Yaskawa INFORM job: R1_W27-A3(90,0)OK-KM.JBI

/JOB
//NAME R1_W27-A3(90,0)OK-KM
///FOLDERNAME KRIS-SCIANA
//POS
///NPOS 39,39,0,3,0,0
///TOOL 0
///POSTYPE PULSE
///PULSE
C00000=28952,8585,-18317,-13996,70208,35679
C00001=71005,-6773,-21567,22823,106593,44775
C00002=117043,42996,63636,80074,76806,36548
C00003=119925,40522,60971,80546,74909,36908
C00004=120979,40510,60955,80742,74190,36976
C00005=121620,40526,60973,80863,73749,37016
C00006=120979,40510,60955,80742,74190,36976
C00007=120972,47430,68505,81028,73985,36463
C00008=120975,44790,65593,80913,74065,36669
C00009=119925,40522,60971,80546,74909,36908
C00010=117043,28525,29392,77595,79872,42812
C00011=119217,29213,30072,77642,78317,42963
C00012=118591,29142,41659,90629,77759,36862
C00013=119665,29075,41592,90781,76989,36871
C00014=118591,29142,41659,90629,77759,36862
C00015=119139,32499,45041,90778,77358,36699
C00016=118591,29142,41659,90629,77759,36862
C00017=117792,30891,31745,84274,86418,41418
C00018=115072,-13134,-7135,52375,63390,45207
C00019=116472,-2069,1649,51986,62773,45649
C00020=119056,6654,11865,54723,60280,45496
C00021=120221,1002,3727,51035,60853,46679
C00022=118976,344,2628,51184,61768,46509
C00023=114063,10407,25128,70575,62115,41682
C00024=112190,-3493,21544,75414,62330,39001
C00025=112095,-4963,21051,75629,62268,38767
C00026=109884,-10292,2975,62963,64916,42297
C00027=110682,-7799,62,53762,64868,43520
C00028=112905,-37925,-18654,59494,39923,-31745
C00029=119033,-32806,-15367,56336,36549,-29573
C00030=103409,10299,29788,79828,70646,-39016
C00031=118213,-31916,-14769,56613,37088,-29774
C00032=119040,-32554,-15197,56304,36559,-29555
C00033=101836,30280,52112,81952,79109,-40621
C00034=100971,47035,98169,91258,69327,-49643
C00035=93737,11259,49117,86061,72646,-45987
C00036=78961,-66055,-35758,60750,43436,-32907
C00037=20797,37541,-3335,35327,72696,-61186
C00038=29399,116943,32129,-7323,87105,-68619
BC00000=188265,1301853,894037
BC00001=296251,1242662,815779
BC00002=395849,1188070,743600
BC00003=395849,1188070,743600
BC00004=395849,1188070,743600
BC00005=395849,1188070,743600
BC00006=395849,1188070,743600
BC00007=395849,1188070,743600
BC00008=395849,1188070,743600
BC00009=395849,1188070,743600
BC00010=395849,1188070,743600
BC00011=395849,1188070,727654
BC00012=394310,1188070,721275
BC00013=394310,1188070,721275
BC00014=394310,1188070,721275
BC00015=394310,1188070,721275
BC00016=394310,1188070,721275
BC00017=395849,1177175,737022
BC00018=360898,1188070,902203
BC00019=357567,1188070,879539
BC00020=356337,1188069,883137
BC00021=356235,1188070,870473
BC00022=356235,1188070,870473
BC00023=356285,1188070,883286
BC00024=356285,1188070,883285
BC00025=356285,1188070,883285
BC00026=356318,1188070,883506
BC00027=360948,1188070,915014
BC00028=346658,1188070,806607
BC00029=342406,1188070,804445
BC00030=341079,1188070,803770
BC00031=340706,1188070,803580
BC00032=340706,1188070,803580
BC00033=340706,1188070,653450
BC00034=340706,1188070,803580
BC00035=341062,1188070,799461
BC00036=346492,1188070,736766
BC00037=227280,1187761,922106
BC00038=106915,1318361,1048473
///POSTYPE BASE
///RECTAN
///RCONF 0,0,0,0,0,0,0,0,0,0,0,0,0,0,0,0,0,0,0,0,0,0,0,0
P00006=0.222,-3.123,-1.508,0.0000,0.0000,0.0000
P00025=-2.003,0.006,0.728,0.0000,0.0000,0.0000
P00026=0.562,-0.002,-0.337,0.0000,0.0000,0.0000
//INST
///DATE 2024/07/29 20:46
///ATTR SC,RW
///GROUP1 RB1,BS1
NOP
SFTOF
MOVJ C00000 BC00000 VJ=100.00
MOVJ C00001 BC00001 VJ=100.00
MOVL C00002 BC00002 V=1000.0
MOVL C00003 BC00003 V=250.0
MOVL C00004 BC00004 V=100.0
REFP 3 C00005 BC00005
CALL JOB:SEARCH-R1
SET P026 P006
SFTON P026
MOVL C00006 BC00006 V=60.0
REFP 3 C00007 BC00007
CALL JOB:SEARCH-R1
SET P026 P006
SFTON P026
MOVL C00008 BC00008 V=60.0
MOVL C00009 BC00009 V=166.7
SFTOF
MOVL C00010 BC00010 V=1000.0
MOVL C00011 BC00011 V=250.0
MOVL C00012 BC00012 V=100.0
REFP 3 C00013 BC00013
CALL JOB:SEARCH-R1
SET P025 P006
SFTON P025
MOVL C00014 BC00014 V=100.0
REFP 3 C00015 BC00015
CALL JOB:SEARCH-R1
SET P025 P006
SFTON P025
MOVL C00016 BC00016 V=100.0
MOVL C00017 BC00017 V=166.7
'Path VIA1038
SFTOF
'Path W998
SFTOF
SFTON P025
MOVJ C00018 BC00018 VJ=100.00
MOVJ C00019 BC00019 VJ=100.00
MOVL C00020 BC00020 V=100.0 PL=0
REFP 1 C00021 BC00021
REFP 2 C00022 BC00022
MACRO1 MJ#(0) ARGF7
ARCON
MOVL C00023 BC00023 V=10.0
MOVL C00024 BC00024 V=11.2
MOVL C00025 BC00025 V=11.2
ARCOF
MOVL C00026 BC00026 V=166.7
MOVL C00027 BC00027 V=166.7
SFTOF
'Path W999
SFTOF
SFTON P025
MOVJ C00028 BC00028 VJ=100.00
MOVJ C00029 BC00029 VJ=100.00
MOVL C00030 BC00030 V=250.0 PL=0
REFP 1 C00031 BC00031
REFP 2 C00032 BC00032
MACRO1 MJ#(0) ARGF7
ARCON
SFTON P026
MOVL C00033 BC00033 V=10.8
ARCOF
MOVL C00034 BC00034 V=250.0
MOVL C00035 BC00035 V=250.0
MOVJ C00036 BC00036 VJ=100.00
SFTOF
MOVJ C00037 BC00037 VJ=100.00
MOVJ C00038 BC00038 VJ=100.00
END
